(* IEC 61131-3 sources: CodesysTest/alpha/export/Device.dev/Plc Logic/Application/FBs/Motors/Applied Motion/FB_AppliedMotionBagDeliveryMotor.pou, 1 file *)

(* ---- SendParameters.m.st ---- *)
(*#-#-#-#-#-#-#-#-#-#---Declaration---#-#-#-#-#-#-#-#-#-#-#-#-#*)

METHOD SendParameters
VAR_INPUT
    reverseSpeed : DINT;

END_VAR
(*#-#-#-#-#-#-#-#-#-#---Implementation---#-#-#-#-#-#-#-#-#-#-#-#-#*)
